(* GVL30_DiagnosticEtherCAT *)
{attribute 'TcContextName' := 'PlcTask'}
VAR_GLOBAL

	fbDiagnosticEtherCAT					:FB_DiagnosticEtherCAT;

END_VAR
(* End *)

(* stored: Version 1.1.0.1, ProductVersion 3.1.4020.3
   GVL GVL30_DiagnosticEtherCAT: Id {60ddb16b-c747-4977-a348-8f2aff42e458} *)
